(* PLC project Untitled1, Beckhoff Automation GmbH TF6420 Database Server Query Analyser 1.0.0.0 *)
(* stored: creationDateTime 2021-07-21T09:10:26, modificationDateTime 2021-07-21T09:10:26 *)

TYPE ST_SelectStruct : STRUCT
  id : LINT;
  sName : STRING(255);
  bIsActive : ARRAY[0..255] OF BYTE;
  bIsAcknowledged : ARRAY[0..255] OF BYTE;
  tActiveStartTime : STRING(255);
  tAckTime : STRING(255);
  tClearedTime : STRING(255);
  uiRepeatCount : DINT;
  sAlarmText : STRING(255);
END_STRUCT;
END_TYPE
